// TIA Portal V19 export
DATA_BLOCK "HYST AND TEMP CUTOFF  DB"   // DB13
{ S7_Optimized_Access := 'TRUE' }
// stored: MemoryReserve 100
   VAR RETAIN
      "MAN SET" : Struct
         "SYRUP MFG_TEMP" : Real;
         "SYRUP MFG_COOLING" : Real;
         "SYRUP MFG_VACCUM" : Real;
         "SYRUP MFG_LOAD CELL" : Real;
         "MFG MOVE PV LOAD CELL" : Real;
         PREMIXING_TEMP : Real;
         PREMIXING_COOLING : Real;
         PREMIXING_VACCUM : Real;
         "PREMIXING_LOAD CELL" : Real;
         "PREMIXING MOVE PV LOAD CELL" : Real;
         SUGAR_TEMP : Real;
         SUGAR_VACCUM : Real;
         "SUGAR_LOAD CELL" : Real;
         "SUGAR MOVE PV LOAD CELL" : Real;
      END_STRUCT;
      "MAIN SET PARA" : Struct
         "SYRUP MFG_TEMP" : Real;
         "SYRUP MFG_COOLING" : Real;
         "SYRUP MFG_VACCUM" : Real;
         "SYRUP MFG_LOAD CELL" : Real;
         "AUTO MFG_LOAD CELL" : Real;
         PREMIXING_TEMP : Real;
         PREMIXING_COOING : Real;
         PREMIXING_VACCUM : Real;
         "PREMIXING_LOAD CELL" : Real;
         "AUTO PREMIXING_LOAD CELL" : Real;
         SUGAR_TEMP : Real;
         SUGAR_VACCUM : Real;
         "SUGAR_LOAD CELL" : Real;
         "AUTO SUGAR_LOAD CELL" : Real;
      END_STRUCT;
      "HYSTERISIS SUB" : Struct
         "SYRUP MFG_TEMP" : Real;
         "SYRUP MFG_COOLING" : Real;
         "SYRUP MFG_VACCUM" : Real;
         "SYRUP MFG_LOAD CELL" : Real;
         PREMIXING_TEMP : Real;
         PREMIXING_COOLING : Real;
         PREMIXING_VACCUM : Real;
         "PREMIXING_LOAD CELL" : Real;
         SUGAR_TEMP : Real;
         SUGAR_VACCUM : Real;
         "SUGAR_LOAD CELL" : Real;
      END_STRUCT;
      "HYSTERISIS NEW_VALUE" : Struct
         "SYRUP MFG_TEMP" : Real;
         "SYRUP MFG_COOLING" : Real;
         "SYRUP MFG_VACCUM" : Real;
         "SYRUP MFG_LOAD CELL" : Real;
         "AUTO MFG_LOAD CELL" : Real;
         PREMIXING_TEMP : Real;
         PREMIXING_COOLING : Real;
         PREMIXING_VACCUM : Real;
         "PREMIXING_LOAD CELL" : Real;
         "AUTO PREMIXING_LOAD CELL" : Real;
         SUGAR_TEMP : Real;
         SUGAR_VACCUM : Real;
         "SUGAR_LOAD CELL" : Real;
         "AUTO SUGAR_LOAD CELL" : Real;
      END_STRUCT;
      "MFG CALCULATE PV" : Real;
      "PREMIXING CALCULATE PV" : Real;
      "SUGAR CALCULATE PV" : Real;
      "AUTO SET" : Struct
         MFG_TEMP : Real;
         MFG_COOLING : Real;
         MFG_VACCUM : Real;
         "MFG_LOAD CELL" : Real;
         "MFG LOAD CELL FOR TRANSFER" : Real;
         PREMIXING_TEMP : Real;
         PREMIXING_COOLING : Real;
         PREMIXING_VACCUM : Real;
         "PREMIXING_LOAD CELL" : Real;
         SUGAR_TEMP : Real;
         SUGAR_VACCUM : Real;
         "SUGAR_LOAD CELL" : Real;
      END_STRUCT;
      "AUTO MAIN SET PARAMETER" : Struct
         "MFG LOAD CELL" : Real;
         "PREMIXING LOAD CELL" : Real;
         "SUGAR LOAD CELL" : Real;
      END_STRUCT;
      "AUTO NEW VALUE" : Struct
         "MFG LOAD CELL" : Real;
         "PREMIXING LOAD CELL" : Real;
         "SUGAR LOAD CELL" : Real;
      END_STRUCT;
      "AUTO MOVE PV" : Struct
         "MFG_LOAD CELL" : Real;
         "PREMIXING_LOAD CELL" : Real;
         "SUGAR_LOAD CELL" : Real;
      END_STRUCT;
   END_VAR
   VAR
      "MIAN MFG TEMP MIN" : Real;
      "MIAN MFG TEMP MAX" : Real;
   END_VAR
BEGIN
END_DATA_BLOCK
